FUNCTION rt_ceild_1 : LREAL
VAR_INPUT
	u: LREAL;
END_VAR
VAR
END_VAR


rt_ceild := DINT_TO_LREAL(TRUNC(u));

IF u = rt_ceild THEN 
    rt_ceild := u;
ELSIF u >= 0.0 THEN 
    rt_ceild := rt_ceild + 1.0;
END_IF;

END_FUNCTION

(* stored: Version 1.1.0.1, ProductVersion 3.1.4024.12
   POU rt_ceild_1: Id {3065b5b4-c09b-4eb8-99d7-d73a8e8c680b}, SpecialFunc None *)
